// TIA Portal V17 export
// export: Created 2025-03-07T09:24:17.007555Z, ExportSetting WithDefaults, DisplayName Totally Integrated Automation Portal, DisplayVersion V17 Update 8, DisplayName TIA Portal Openness, DisplayVersion V17 Update 8, DisplayName TIA Portal Version Control Interface, DisplayVersion V17, DisplayName SINAMICS Startdrive Advanced, DisplayVersion V17 SP2, DisplayName SINAMICS Startdrive G110M, G120, G120C, G120D, G120P, G115D, DisplayVersion V17 SP2, DisplayName SINAMICS Startdrive G130, G150, S120, S150, SINAMICS MV, S210, DisplayVersion V17 SP2, DisplayName STEP 7 Professional, DisplayVersion V17 Update 8, DisplayName SINUMERIK ONE STEP 7 Toolbox, DisplayVersion V17 Update 12, DisplayName SINUMERIK 840D sl STEP 7 Toolbox, DisplayVersion V17 Update 12, DisplayName STEP 7 Safety, DisplayVersion V17 Update 6, DisplayName WinCC Advanced, DisplayVersion V17 Update 8
DATA_BLOCK "DB22141_PRESSURE_FEEDER_2_HOPPER_1_UNIT_02"   // DB22141
{ DB_Accessible_From_OPC_UA := 'FALSE' }
VERSION : 0.1
// stored: AutoNumber false, DBAccessibleFromOPCUA false, DBAccessibleFromWebserver true, InstanceOfName FB22101_PRESSURE_SENSOR, InstanceOfType FB
"FB22101_PRESSURE_SENSOR"
   // VAR_INPUT
   //    iINPUT_VALUE : Int;
   //    iCLEAR_INTERNAL_LOG : Bool;
   //    iSAVE_MAX_PRESSURE : Bool;
   // END_VAR
   // VAR_OUTPUT
   //    oWARNING_LIMIT : Bool;
   //    oERROR_LIMIT : Bool;
   // END_VAR
   // VAR
   //    OUTPUT : Struct
   //       VALUE : Real;
   //    END_STRUCT;
   //    INPUT_SETTINGS : Struct
   //       DIV_VALUE : Real;
   //       NORM_MIN_VALUE : DInt;
   //       NORM_MAX_VALUE : DInt;
   //       LOW_RANGE : Real := -1.0;
   //       HIGH_RANGE : Real := 1.0;
   //       IS_ANALOG_VALUE : Bool := true;
   //       UNIT_NUMBER : Int := 2;
   //       HOPPER_NUMBER : Int := 3;
   //    END_STRUCT;
   //    ALARMS_SETTINGS : Struct
   //       WARN_LIM_LOW : Real;
   //       ERROR_LIM_LOW : Real;
   //       WARN_LIM_HIGH : Real;
   //       ERROR_LIM_HIGH : Real;
   //       ERROR_CONFIGURATION : Bool;
   //    END_STRUCT;
   //    LOG : Struct
   //       DATE_MAX_PRESSURE : Date_And_Time;
   //       "VALUE_MAX PRESSURE" : Real;
   //    END_STRUCT;
   //    INTERNAL : Struct
   //       AUXILIARY_TRIGGER : Bool;
   //    END_STRUCT;
   // END_VAR
BEGIN
END_DATA_BLOCK
